// TIA Portal V18 export
FUNCTION "Flush sequences" : Void   // FC17, LAD
{ S7_Optimized_Access := 'TRUE' }
VERSION : 0.1
// stored: AutoNumber true, IsIECCheckEnabled false, SetENOAutomatically false, UDAEnableTagReadback false
   VAR_TEMP
      temp1 : Bool;
      temp2 : Bool;
   END_VAR
   VAR_TEMP   // added for the SCL form of the ladder/FBD networks
      _w1 : Bool;
      _w2 : Bool;
   END_VAR
BEGIN

REGION Network 1 (SCL)
   IF "Function Flush".Selection = 0 THEN
       "Functions"."flush selection"."Flush A selected" := true;
       "Functions"."flush selection"."Flush B selected" := false;
       "Pump & Flowrate"."Flush Maximum Flowrate" := "Pump & Flowrate".capacity."Pump A";
       "Pump & Flowrate"."Flush minimum Flowrate" := "Pump & Flowrate".capacity."Pump A" * 0.10;
       "Function Flush"."Input A"."set time in sec" := REAL_TO_DINT(("Function Flush"."Input A"."set qty" / "Function Flush"."Input A"."set flowrate") * 60.0);
   ELSE
       "Functions"."flush selection"."Flush A selected" := false;
       "Functions"."flush selection"."Flush B selected" := true;
       "Pump & Flowrate"."Flush Maximum Flowrate" := "Pump & Flowrate".capacity."pump B";
       "Pump & Flowrate"."Flush minimum Flowrate" := "Pump & Flowrate".capacity."pump B" * 0.10;
       "Function Flush"."Input B"."set time in sec" := REAL_TO_DINT(("Function Flush"."Input B"."set qty" / "Function Flush"."Input B"."set flowrate") * 60.0);
   END_IF;
END_REGION

REGION Network 2: Flush A sequences
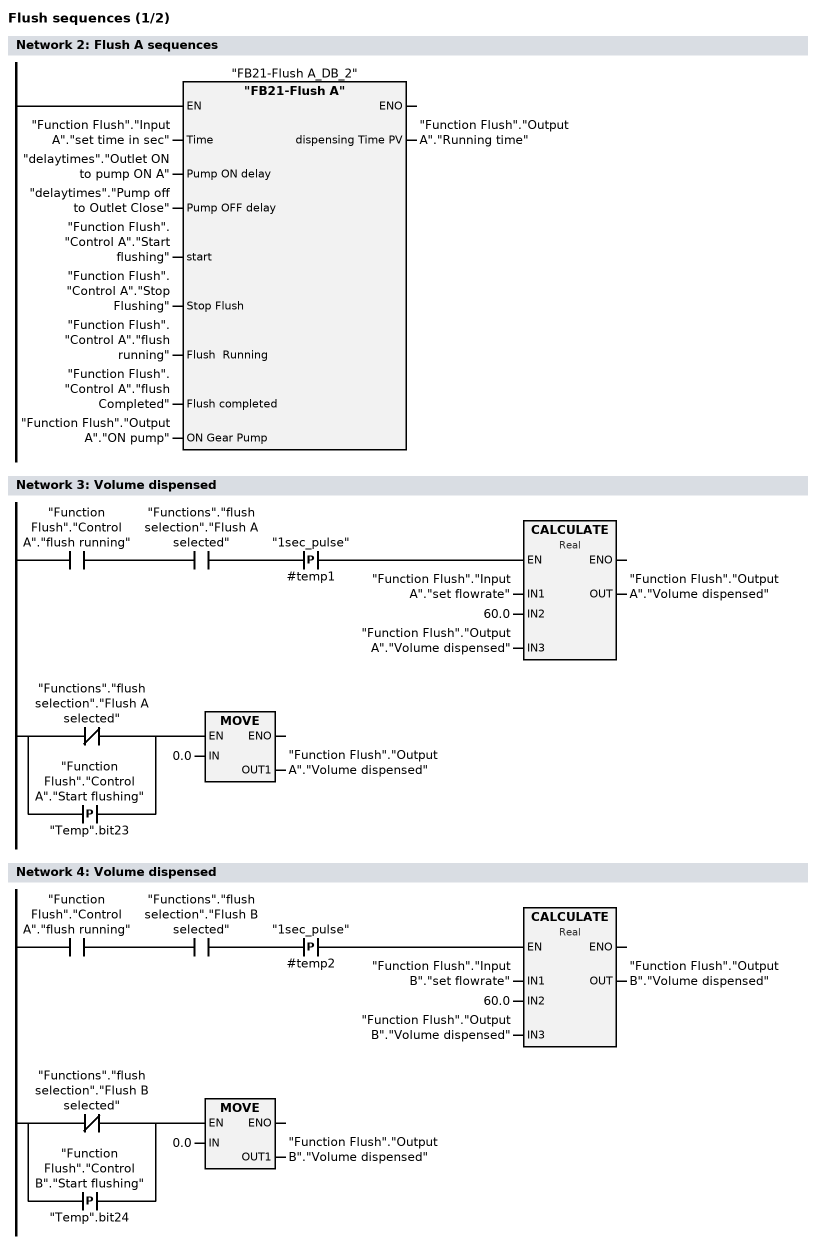
   RUNG wire#powerrail
      "FB21-Flush A_DB_2"("Time" := "Function Flush"."Input A"."set time in sec", "Pump ON delay" := "delaytimes"."Outlet ON to pump ON A", "Pump OFF delay" := "delaytimes"."Pump off to Outlet Close", start := "Function Flush"."Control A"."Start flushing", "Stop Flush" := "Function Flush"."Control A"."Stop Flushing", "Flush  Running" := "Function Flush"."Control A"."flush running", "Flush completed" := "Function Flush"."Control A"."flush Completed", "ON Gear Pump" := "Function Flush"."Output A"."ON pump", "dispensing Time PV" => "Function Flush"."Output A"."Running time")
   END_RUNG
   // the same network as SCL:
   "FB21-Flush A_DB_2"("Time" := "Function Flush"."Input A"."set time in sec",   // "FB21-Flush A"
                       "Pump ON delay" := "delaytimes"."Outlet ON to pump ON A",
                       "Pump OFF delay" := "delaytimes"."Pump off to Outlet Close",
                       start := "Function Flush"."Control A"."Start flushing",
                       "Stop Flush" := "Function Flush"."Control A"."Stop Flushing",
                       "Flush  Running" := "Function Flush"."Control A"."flush running",
                       "Flush completed" := "Function Flush"."Control A"."flush Completed",
                       "ON Gear Pump" := "Function Flush"."Output A"."ON pump",
                       "dispensing Time PV" => "Function Flush"."Output A"."Running time");
END_REGION

REGION Network 3: Volume dispensed
   RUNG wire#powerrail
      Contact( "Function Flush"."Control A"."flush running" )
      Contact( "Functions"."flush selection"."Flush A selected" )
      P_Contact(operand := "1sec_pulse", bit := #temp1)
      { S7_Templates := "SrcType := Real"; S7_Expression := "(IN1/IN2)+IN3" } Calculate(in1 := "Function Flush"."Input A"."set flowrate", in2 := 60.0, in3 := "Function Flush"."Output A"."Volume dispensed", out => "Function Flush"."Output A"."Volume dispensed")
   END_RUNG
   RUNG wire#powerrail
      I_Contact( "Functions"."flush selection"."Flush A selected" )
      wire#w1
      Move(in := 0.0, out1 => "Function Flush"."Output A"."Volume dispensed")
   END_RUNG
   RUNG wire#powerrail
      P_Contact(operand := "Function Flush"."Control A"."Start flushing", bit := "Temp".bit23)
   END_RUNG wire#w1
   // the same network as SCL:
   #_w1 := "Function Flush"."Control A"."flush running" AND "Functions"."flush selection"."Flush A selected" AND "1sec_pulse" AND NOT #temp1;   // rising edge of "1sec_pulse"
   #temp1 := "1sec_pulse";
   IF #_w1 THEN
       "Function Flush"."Output A"."Volume dispensed" := ("Function Flush"."Input A"."set flowrate"/60.0)+"Function Flush"."Output A"."Volume dispensed";
   END_IF;
   #_w2 := "Function Flush"."Control A"."Start flushing" AND NOT "Temp".bit23;   // rising edge of "Function Flush"."Control A"."Start flushing"
   "Temp".bit23 := "Function Flush"."Control A"."Start flushing";
   IF NOT "Functions"."flush selection"."Flush A selected" OR #_w2 THEN
       "Function Flush"."Output A"."Volume dispensed" := 0.0;
   END_IF;
END_REGION

REGION Network 4: Volume dispensed
   RUNG wire#powerrail
      Contact( "Function Flush"."Control A"."flush running" )
      Contact( "Functions"."flush selection"."Flush B selected" )
      P_Contact(operand := "1sec_pulse", bit := #temp2)
      { S7_Templates := "SrcType := Real"; S7_Expression := "(IN1/IN2)+IN3" } Calculate(in1 := "Function Flush"."Input B"."set flowrate", in2 := 60.0, in3 := "Function Flush"."Output B"."Volume dispensed", out => "Function Flush"."Output B"."Volume dispensed")
   END_RUNG
   RUNG wire#powerrail
      I_Contact( "Functions"."flush selection"."Flush B selected" )
      wire#w1
      Move(in := 0.0, out1 => "Function Flush"."Output B"."Volume dispensed")
   END_RUNG
   RUNG wire#powerrail
      P_Contact(operand := "Function Flush"."Control B"."Start flushing", bit := "Temp".bit24)
   END_RUNG wire#w1
   // the same network as SCL:
   #_w1 := "Function Flush"."Control A"."flush running" AND "Functions"."flush selection"."Flush B selected" AND "1sec_pulse" AND NOT #temp2;   // rising edge of "1sec_pulse"
   #temp2 := "1sec_pulse";
   IF #_w1 THEN
       "Function Flush"."Output B"."Volume dispensed" := ("Function Flush"."Input B"."set flowrate"/60.0)+"Function Flush"."Output B"."Volume dispensed";
   END_IF;
   #_w2 := "Function Flush"."Control B"."Start flushing" AND NOT "Temp".bit24;   // rising edge of "Function Flush"."Control B"."Start flushing"
   "Temp".bit24 := "Function Flush"."Control B"."Start flushing";
   IF NOT "Functions"."flush selection"."Flush B selected" OR #_w2 THEN
       "Function Flush"."Output B"."Volume dispensed" := 0.0;
   END_IF;
END_REGION

REGION Network 5: Set Time In hmi
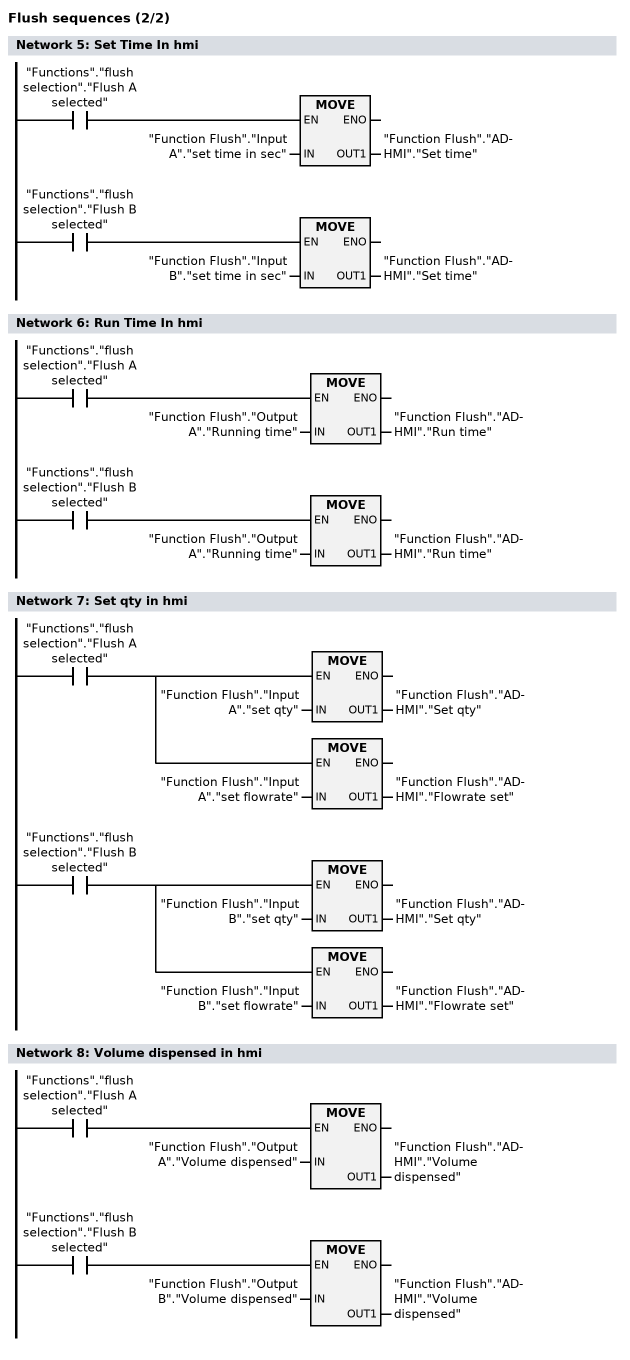
   RUNG wire#powerrail
      Contact( "Functions"."flush selection"."Flush A selected" )
      Move(in := "Function Flush"."Input A"."set time in sec", out1 => "Function Flush"."AD-HMI"."Set time")
   END_RUNG
   RUNG wire#powerrail
      Contact( "Functions"."flush selection"."Flush B selected" )
      Move(in := "Function Flush"."Input B"."set time in sec", out1 => "Function Flush"."AD-HMI"."Set time")
   END_RUNG
   // the same network as SCL:
   IF "Functions"."flush selection"."Flush A selected" THEN
       "Function Flush"."AD-HMI"."Set time" := "Function Flush"."Input A"."set time in sec";
   END_IF;
   IF "Functions"."flush selection"."Flush B selected" THEN
       "Function Flush"."AD-HMI"."Set time" := "Function Flush"."Input B"."set time in sec";
   END_IF;
END_REGION

REGION Network 6: Run Time In hmi
   RUNG wire#powerrail
      Contact( "Functions"."flush selection"."Flush A selected" )
      Move(in := "Function Flush"."Output A"."Running time", out1 => "Function Flush"."AD-HMI"."Run time")
   END_RUNG
   RUNG wire#powerrail
      Contact( "Functions"."flush selection"."Flush B selected" )
      Move(in := "Function Flush"."Output A"."Running time", out1 => "Function Flush"."AD-HMI"."Run time")
   END_RUNG
   // the same network as SCL:
   IF "Functions"."flush selection"."Flush A selected" THEN
       "Function Flush"."AD-HMI"."Run time" := "Function Flush"."Output A"."Running time";
   END_IF;
   IF "Functions"."flush selection"."Flush B selected" THEN
       "Function Flush"."AD-HMI"."Run time" := "Function Flush"."Output A"."Running time";
   END_IF;
END_REGION

REGION Network 7: Set qty in hmi
   RUNG wire#powerrail
      Contact( "Functions"."flush selection"."Flush A selected" )
      wire#w1
      Move(in := "Function Flush"."Input A"."set qty", out1 => "Function Flush"."AD-HMI"."Set qty")
   END_RUNG
   RUNG wire#w1
      Move(in := "Function Flush"."Input A"."set flowrate", out1 => "Function Flush"."AD-HMI"."Flowrate set")
   END_RUNG
   RUNG wire#powerrail
      Contact( "Functions"."flush selection"."Flush B selected" )
      wire#w2
      Move(in := "Function Flush"."Input B"."set qty", out1 => "Function Flush"."AD-HMI"."Set qty")
   END_RUNG
   RUNG wire#w2
      Move(in := "Function Flush"."Input B"."set flowrate", out1 => "Function Flush"."AD-HMI"."Flowrate set")
   END_RUNG
   // the same network as SCL:
   IF "Functions"."flush selection"."Flush A selected" THEN
       "Function Flush"."AD-HMI"."Set qty" := "Function Flush"."Input A"."set qty";
       "Function Flush"."AD-HMI"."Flowrate set" := "Function Flush"."Input A"."set flowrate";
   END_IF;
   IF "Functions"."flush selection"."Flush B selected" THEN
       "Function Flush"."AD-HMI"."Set qty" := "Function Flush"."Input B"."set qty";
       "Function Flush"."AD-HMI"."Flowrate set" := "Function Flush"."Input B"."set flowrate";
   END_IF;
END_REGION

REGION Network 8: Volume dispensed in hmi
   RUNG wire#powerrail
      Contact( "Functions"."flush selection"."Flush A selected" )
      Move(in := "Function Flush"."Output A"."Volume dispensed", out1 => "Function Flush"."AD-HMI"."Volume dispensed")
   END_RUNG
   RUNG wire#powerrail
      Contact( "Functions"."flush selection"."Flush B selected" )
      Move(in := "Function Flush"."Output B"."Volume dispensed", out1 => "Function Flush"."AD-HMI"."Volume dispensed")
   END_RUNG
   // the same network as SCL:
   IF "Functions"."flush selection"."Flush A selected" THEN
       "Function Flush"."AD-HMI"."Volume dispensed" := "Function Flush"."Output A"."Volume dispensed";
   END_IF;
   IF "Functions"."flush selection"."Flush B selected" THEN
       "Function Flush"."AD-HMI"."Volume dispensed" := "Function Flush"."Output B"."Volume dispensed";
   END_IF;
END_REGION
END_FUNCTION
